Yaskawa INFORM job: EXAMPLE.JBI

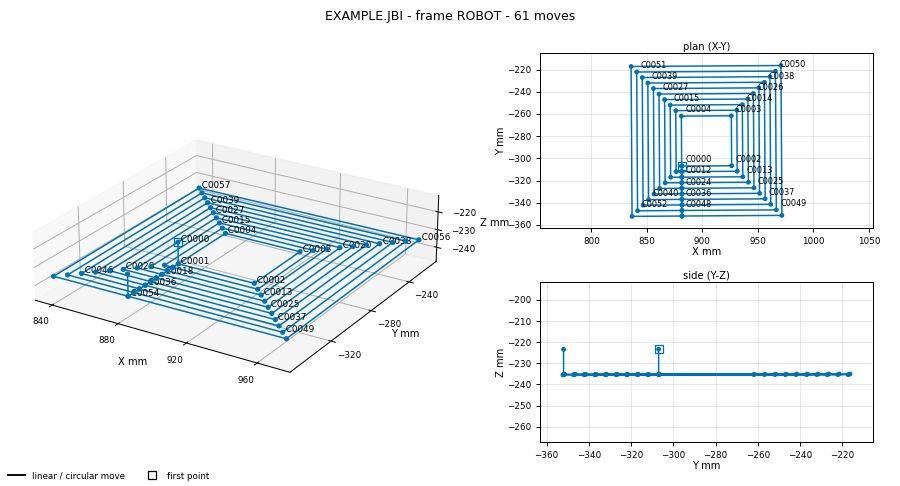
[picture p0: tool path of EXAMPLE.JBI in frame ROBOT, 61 of 61 moves have a stored position in this frame; points joined in program order, loops and branches not executed]
/JOB
//NAME GHTEST4
//POS
///NPOS 61,0,0,0,0,0
///TOOL 1
///POSTYPE ROBOT
///RECTAN
///RCONF 0,0,0,0,0
C0000=881.358,-306.982,-223.343,-90.00,90.00,-90.00
C0001=881.385,-306.971,-235.343,-90.00,90.00,-90.00
C0002=926.384,-306.682,-235.241,-90.00,90.00,-90.00
C0003=926.095,-261.683,-235.198,-90.00,90.00,-90.00
C0004=881.096,-261.972,-235.301,-90.00,90.00,-90.00
C0005=881.385,-306.971,-235.343,-90.00,90.00,-90.00
C0006=881.417,-311.971,-235.348,-90.00,90.00,-90.00
C0007=931.416,-311.649,-235.234,-90.00,90.00,-90.00
C0008=931.062,-256.651,-235.182,-90.00,90.00,-90.00
C0009=876.064,-257.004,-235.307,-90.00,90.00,-90.00
C0010=876.417,-312.003,-235.36,-90.00,90.00,-90.00
C0011=881.417,-311.971,-235.348,-90.00,90.00,-90.00
C0012=881.449,-316.971,-235.353,-90.00,90.00,-90.00
C0013=936.448,-316.617,-235.228,-90.00,90.00,-90.00
C0014=936.03,-251.619,-235.166,-90.00,90.00,-90.00
C0015=871.032,-252.036,-235.314,-90.00,90.00,-90.00
C0016=871.449,-317.035,-235.376,-90.00,90.00,-90.00
C0017=881.449,-316.971,-235.353,-90.00,90.00,-90.00
C0018=881.481,-321.97,-235.358,-90.00,90.00,-90.00
C0019=941.48,-321.585,-235.221,-90.00,90.00,-90.00
C0020=940.998,-246.587,-235.15,-90.00,90.00,-90.00
C0021=866.0,-247.068,-235.32,-90.00,90.00,-90.00
C0022=866.482,-322.067,-235.392,-90.00,90.00,-90.00
C0023=881.481,-321.97,-235.358,-90.00,90.00,-90.00
C0024=881.514,-326.97,-235.362,-90.00,90.00,-90.00
C0025=946.512,-326.553,-235.215,-90.00,90.00,-90.00
C0026=945.966,-241.555,-235.134,-90.00,90.00,-90.00
C0027=860.968,-242.101,-235.327,-90.00,90.00,-90.00
C0028=861.514,-327.099,-235.408,-90.00,90.00,-90.00
C0029=881.514,-326.97,-235.362,-90.00,90.00,-90.00
C0030=881.546,-331.97,-235.367,-90.00,90.00,-90.00
C0031=951.544,-331.521,-235.208,-90.00,90.00,-90.00
C0032=950.933,-236.523,-235.117,-90.00,90.00,-90.00
C0033=855.936,-237.133,-235.334,-90.00,90.00,-90.00
C0034=856.546,-332.131,-235.424,-90.00,90.00,-90.00
C0035=881.546,-331.97,-235.367,-90.00,90.00,-90.00
C0036=881.578,-336.97,-235.372,-90.00,90.00,-90.00
C0037=956.576,-336.488,-235.201,-90.00,90.00,-90.00
C0038=955.901,-231.491,-235.101,-90.00,90.00,-90.00
C0039=850.904,-232.165,-235.34,-90.00,90.00,-90.00
C0040=851.579,-337.163,-235.44,-90.00,90.00,-90.00
C0041=881.578,-336.97,-235.372,-90.00,90.00,-90.00
C0042=881.61,-341.97,-235.377,-90.00,90.00,-90.00
C0043=961.608,-341.456,-235.195,-90.00,90.00,-90.00
C0044=960.869,-226.458,-235.085,-90.00,90.00,-90.00
C0045=845.872,-227.197,-235.347,-90.00,90.00,-90.00
C0046=846.611,-342.195,-235.456,-90.00,90.00,-90.00
C0047=881.61,-341.97,-235.377,-90.00,90.00,-90.00
C0048=881.642,-346.97,-235.382,-90.00,90.00,-90.00
C0049=966.64,-346.424,-235.188,-90.00,90.00,-90.00
C0050=965.837,-221.426,-235.069,-90.00,90.00,-90.00
C0051=840.84,-222.23,-235.353,-90.00,90.00,-90.00
C0052=841.643,-347.227,-235.473,-90.00,90.00,-90.00
C0053=881.642,-346.97,-235.382,-90.00,90.00,-90.00
C0054=881.674,-351.97,-235.386,-90.00,90.00,-90.00
C0055=971.672,-351.392,-235.181,-90.00,90.00,-90.00
C0056=970.804,-216.394,-235.053,-90.00,90.00,-90.00
C0057=835.808,-217.262,-235.36,-90.00,90.00,-90.00
C0058=836.675,-352.259,-235.489,-90.00,90.00,-90.00
C0059=881.674,-351.97,-235.386,-90.00,90.00,-90.00
C0060=881.647,-351.981,-223.386,-90.00,90.00,-90.00
//INST
///DATE 2015/05/22 15:03
///ATTR SC,RW,RJ
////FRAME ROBOT
///GROUP1 RB1
NOP
MOVL C0000 V=50
MOVL C0001 V=50
DOUT OT#(121) ON
MOVL C0002 V=50
MOVL C0003 V=50
MOVL C0004 V=50
MOVL C0005 V=50
MOVL C0006 V=50
MOVL C0007 V=50
MOVL C0008 V=50
MOVL C0009 V=50
MOVL C0010 V=50
MOVL C0011 V=50
MOVL C0012 V=50
MOVL C0013 V=50
MOVL C0014 V=50
MOVL C0015 V=50
MOVL C0016 V=50
MOVL C0017 V=50
MOVL C0018 V=50
MOVL C0019 V=50
MOVL C0020 V=50
MOVL C0021 V=50
MOVL C0022 V=50
MOVL C0023 V=50
MOVL C0024 V=50
MOVL C0025 V=50
MOVL C0026 V=50
MOVL C0027 V=50
MOVL C0028 V=50
MOVL C0029 V=50
MOVL C0030 V=50
MOVL C0031 V=50
MOVL C0032 V=50
MOVL C0033 V=50
MOVL C0034 V=50
MOVL C0035 V=50
MOVL C0036 V=50
MOVL C0037 V=50
MOVL C0038 V=50
MOVL C0039 V=50
MOVL C0040 V=50
MOVL C0041 V=50
MOVL C0042 V=50
MOVL C0043 V=50
MOVL C0044 V=50
MOVL C0045 V=50
MOVL C0046 V=50
MOVL C0047 V=50
MOVL C0048 V=50
MOVL C0049 V=50
MOVL C0050 V=50
MOVL C0051 V=50
MOVL C0052 V=50
MOVL C0053 V=50
MOVL C0054 V=50
MOVL C0055 V=50
MOVL C0056 V=50
MOVL C0057 V=50
MOVL C0058 V=50
MOVL C0059 V=50
DOUT OT#(121) OFF
MOVL C0060 V=50
END
